FUNCTION_BLOCK RejectWithMessageAsyncHandler IMPLEMENTS I_AsynchronousRpcHandler
VAR
END_VAR

METHOD Handle
VAR_INPUT
	Parameters : I_Deserializer;
	Response : I_AsynchronousRpcResponse;
END_VAR
VAR
END_VAR
Response.RejectWithError('EXAMPLE_ERROR_CODE','This is the reject message');
END_METHOD

END_FUNCTION_BLOCK

(* stored: Version 1.1.0.1, ProductVersion 3.1.4026.13
   POU RejectWithMessageAsyncHandler: Id {cb9503fc-4aa7-0763-24ec-bc44822dcf7e}, SpecialFunc None
   Method Handle: Id {d1acf3c1-eeda-048f-1f5a-1add869c4d30} *)
